(* IEC 61131-3 sources: Word/plc-course/23-commissioning-and-troubleshooting/labs/starter, 3 files *)

(* ---- 23-1-find-the-bugs.st ---- *)
(* Lab 23-1: Find the bugs - transfer conveyor with jog and jam detection.
   Module 23 (Commissioning and troubleshooting). STARTER - this program is
   complete and it compiles, but the site has reported three faults and the
   acceptance test fails. Run it to see the failures:
     python3 tools/plctest.py 23-commissioning-and-troubleshooting/labs/starter/23-1-find-the-bugs.st
   Copy it to your own folder, find the three bugs and fix them with the
   smallest change that removes each root cause. Don't rewrite the program. *)

PROGRAM TransferConveyor
  VAR (* I/O - addresses follow the OpenPLC convention *)
    StartPB       AT %IX0.0 : BOOL;  (* Start push-button, NO: TRUE while pressed *)
    StopPB_NC     AT %IX0.1 : BOOL;  (* Stop push-button, NC: TRUE while NOT pressed *)
    JogPB         AT %IX0.2 : BOOL;  (* Jog push-button, NO: conveyor runs only while held *)
    JamPE         AT %IX0.3 : BOOL;  (* Jam photo-eye at the discharge: TRUE while the beam is blocked *)
    ResetPB       AT %IX0.4 : BOOL;  (* Fault reset push-button, NO *)
    OverloadOK_NC AT %IX0.5 : BOOL;  (* Motor overload relay auxiliary contact, NC: TRUE while healthy *)
    ConveyorMotor AT %QX0.0 : BOOL;  (* Conveyor motor contactor coil *)
    RunLamp       AT %QX0.1 : BOOL;  (* Green lamp: running in automatic *)
    FaultLamp     AT %QX0.2 : BOOL;  (* Red lamp: a fault is latched *)
  END_VAR
  VAR (* internal *)
    RunLatch : BOOL;  (* automatic run, sealed in by Start *)
    JogRun   : BOOL;  (* jog command *)
    Fault    : BOOL;  (* latched fault: jam or motor overload *)
    JamTimer : TON;   (* photo-eye blocked for too long while running = jam *)
  END_VAR

  (* ---- 1. Jam detection: only needed while the conveyor runs ------------ *)
  IF RunLatch THEN
    JamTimer(IN := JamPE, PT := T#3s);
  END_IF;

  (* ---- 2. Fault latch: set by the cause, reset only when the cause has gone *)
  IF JamTimer.Q OR NOT OverloadOK_NC THEN
    Fault := TRUE;
  ELSIF ResetPB AND NOT JamPE AND OverloadOK_NC THEN
    Fault := FALSE;
  END_IF;

  (* ---- 3. Automatic run: Start seals in, Stop (or a broken stop wire) drops it *)
  RunLatch := (StartPB OR RunLatch) AND StopPB_NC;
  ConveyorMotor := RunLatch AND NOT Fault;

  (* ---- 4. Jog for maintenance: momentary, only when stopped and healthy *)
  JogRun := JogPB AND StopPB_NC AND NOT RunLatch AND NOT Fault;
  ConveyorMotor := JogRun;

  (* ---- 5. Lamps *)
  RunLamp := RunLatch AND NOT Fault;
  FaultLamp := Fault;
END_PROGRAM

CONFIGURATION Config0
  RESOURCE Res0 ON PLC
    TASK MainTask(INTERVAL := T#10ms, PRIORITY := 0);
    PROGRAM Inst0 WITH MainTask : TransferConveyor;
  END_RESOURCE
END_CONFIGURATION

(* ---- 23-2-subtle-faults.st ---- *)
(* Lab 23-2: Subtle faults - drum filling station.
   Module 23 (Commissioning and troubleshooting). STARTER - this program passed
   its bench test and has been running on site for a month. It compiles and it
   mostly works, but the site has reported three faults (see the lab sheet in
   the README) and the acceptance test fails. Run it to see the failures:
     python3 tools/plctest.py 23-commissioning-and-troubleshooting/labs/starter/23-2-subtle-faults.st
   Copy it to your own folder, find the three root causes and fix them. Keep
   every name in the interface table; change as little as you can. *)

TYPE
  E_FillStep : (Idle, Filling, Done);
END_TYPE

PROGRAM DrumFiller
  VAR (* I/O - addresses follow the OpenPLC convention *)
    StartPB       AT %IX0.0 : BOOL;  (* Start push-button, NO *)
    StopPB_NC     AT %IX0.1 : BOOL;  (* Stop push-button, NC: TRUE while NOT pressed *)
    DrumPresentPX AT %IX0.2 : BOOL;  (* Proximity switch: a drum is in position on the scale *)
    WeightRaw     AT %IW0   : INT;   (* Scale transmitter via 4-20 mA input: 0..27648 = 0..300 kg *)
    FillValve     AT %QX0.0 : BOOL;  (* Fill valve solenoid, spring-return: de-energised = closed *)
    DoneLamp      AT %QX0.1 : BOOL;  (* White lamp: drum full, remove it *)
  END_VAR
  VAR (* HMI commands: the HMI writes TRUE, the PLC clears them (momentary) *)
    HmiStartCmd      : BOOL;  (* HMI "Start fill" button *)
    HmiResetCountCmd : BOOL;  (* HMI "Reset shift count" button *)
  END_VAR
  VAR (* HMI display values *)
    Weight_kg : REAL;  (* gross weight on the scale *)
    TotalKg   : DINT;  (* nominal kg filled this shift = DrumCount x 200 kg *)
  END_VAR
  VAR RETAIN (* must survive a power cut *)
    DrumCount : INT;         (* drums filled this shift *)
    FillStep  : E_FillStep;  (* where the sequence is *)
  END_VAR
  VAR (* internal *)
    StartReq : BOOL;
    Tare_kg  : REAL;  (* weight of the empty drum, captured at the start *)
    Net_kg   : REAL;  (* product added so far *)
  END_VAR
  VAR CONSTANT
    TargetNet_kg   : REAL := 200.0;  (* product per drum *)
    EmptyMax_kg    : REAL := 50.0;   (* heavier than this = not an empty drum *)
    DrumNominal_kg : INT := 200;     (* used for the shift total *)
  END_VAR

  (* ---- 0. Housekeeping: HMI buttons are momentary, so the PLC clears them.
     (Added after an HMI lost its connection with a command stuck TRUE.) *)
  HmiStartCmd := FALSE;
  HmiResetCountCmd := FALSE;

  (* ---- 1. Scale: raw counts to kilograms (Module 14) *)
  Weight_kg := INT_TO_REAL(WeightRaw) * 300.0 / 27648.0;

  (* ---- 2. Start request from the panel push-button or the HMI *)
  StartReq := StartPB OR HmiStartCmd;

  (* ---- 3. Fill sequence *)
  CASE FillStep OF
    Idle:
      (* Start only with a healthy stop circuit and an EMPTY drum in place *)
      IF StartReq AND StopPB_NC AND DrumPresentPX AND (Weight_kg < EmptyMax_kg) THEN
        Tare_kg := Weight_kg;
        Net_kg := 0.0;
        FillStep := Filling;
      END_IF;

    Filling:
      Net_kg := Weight_kg - Tare_kg;
      IF NOT StopPB_NC OR NOT DrumPresentPX THEN
        FillStep := Idle;                      (* abort: this drum is not counted *)
      ELSIF Net_kg >= TargetNet_kg THEN
        DrumCount := DrumCount + 1;
        FillStep := Done;
      END_IF;

    Done:
      IF NOT DrumPresentPX THEN            (* full drum taken away *)
        FillStep := Idle;
      END_IF;
  END_CASE;

  (* ---- 4. Shift totals. TotalKg is a DINT, so it cannot overflow. *)
  IF HmiResetCountCmd THEN
    DrumCount := 0;
  END_IF;
  TotalKg := INT_TO_DINT(DrumCount * DrumNominal_kg);

  (* ---- 5. Outputs, written once, from the step *)
  FillValve := (FillStep = Filling);
  DoneLamp := (FillStep = Done);
END_PROGRAM

CONFIGURATION Config0
  RESOURCE Res0 ON PLC
    TASK MainTask(INTERVAL := T#10ms, PRIORITY := 0);
    PROGRAM Inst0 WITH MainTask : DrumFiller;
  END_RESOURCE
END_CONFIGURATION

(* ---- 23-3-io-simulation.st ---- *)
(* Lab 23-3: I/O simulation layer for checkout - transfer pump P-101.
   Module 23 (Commissioning and troubleshooting). STARTER - the types, the
   declarations and the application logic are done for you. Write the
   simulation layer where it says TODO (you may add your own function blocks
   above the program), then run:
     python3 tools/plctest.py 23-commissioning-and-troubleshooting/labs/starter/23-3-io-simulation.st
   Training exercise only: simulation must never bypass a safety function. *)

TYPE
  ST_SimDI : STRUCT
    Enable : BOOL;  (* HMI: put this point into simulation *)
    Value  : BOOL;  (* HMI: simulated value *)
  END_STRUCT;
  ST_SimAI : STRUCT
    Enable : BOOL;  (* HMI: put this point into simulation *)
    Value  : REAL;  (* HMI: simulated value in engineering units *)
  END_STRUCT;
END_TYPE

PROGRAM PumpCheckout
  VAR (* I/O - addresses follow the OpenPLC convention *)
    LSL101_NC AT %IX0.0 : BOOL;  (* LSL-101 low-level switch, NC: TRUE while level is above it *)
    P101RunFB AT %IX0.1 : BOOL;  (* P-101 contactor auxiliary contact: TRUE = running *)
    SimKeySW  AT %IX0.2 : BOOL;  (* key switch "simulation permitted" (commissioning only) *)
    ResetPB   AT %IX0.3 : BOOL;  (* fault reset push-button, NO *)
    LT101Raw  AT %IW0   : INT;   (* LT-101 tank level, 4-20 mA input: 0..27648 = 0..100 % *)
    P101Run   AT %QX0.0 : BOOL;  (* P-101 contactor coil *)
    SimLamp   AT %QX0.1 : BOOL;  (* amber lamp: simulation active *)
    P101Fault AT %QX0.2 : BOOL;  (* red lamp: P-101 failed to start *)
  END_VAR
  VAR (* HMI simulation tags, one structure per point *)
    SimLSL101 : ST_SimDI;
    SimP101FB : ST_SimDI;
    SimLT101  : ST_SimAI;
  END_VAR
  VAR (* processed values: the ONLY input values the application logic uses *)
    LSL101_OK   : BOOL;
    P101Running : BOOL;
    LT101_Pct   : REAL;
  END_VAR
  VAR (* simulation status for the HMI banner *)
    SimActive : BOOL;
    SimCount  : INT;
  END_VAR
  VAR (* internal: add your own variables and FB instances here *)
    PumpDemand : BOOL;
    FbTimer    : TON;
  END_VAR

  (* ==== SIMULATION LAYER ====
     TODO: replace these placeholder lines. For each of the three points, set
     the processed value from the field or from its simulation structure,
     following the lab requirements. Then set SimCount, SimActive and SimLamp. *)
  LSL101_OK := FALSE;
  P101Running := FALSE;
  LT101_Pct := 0.0;
  SimCount := 0;
  SimActive := FALSE;
  SimLamp := FALSE;

  (* ==== APPLICATION LOGIC (given; uses processed values only) ==== *)
  (* Level control with hysteresis: start at 60 %, stop at 20 % *)
  IF LT101_Pct >= 60.0 THEN
    PumpDemand := TRUE;
  ELSIF LT101_Pct <= 20.0 THEN
    PumpDemand := FALSE;
  END_IF;

  (* Start failure: commanded but no running feedback within 2 s *)
  FbTimer(IN := P101Run AND NOT P101Running, PT := T#2s);
  IF FbTimer.Q THEN
    P101Fault := TRUE;
  ELSIF ResetPB THEN
    P101Fault := FALSE;
  END_IF;

  (* Command: demand AND dry-run protection AND no fault *)
  P101Run := PumpDemand AND LSL101_OK AND NOT P101Fault;
END_PROGRAM

CONFIGURATION Config0
  RESOURCE Res0 ON PLC
    TASK MainTask(INTERVAL := T#10ms, PRIORITY := 0);
    PROGRAM Inst0 WITH MainTask : PumpCheckout;
  END_RESOURCE
END_CONFIGURATION
